// TwinCAT 3 PLC project PLC_Project
// ProgramVersion: 3.1.4024.0
// libraries:
//   Tc2_ControllerToolbox, * (Beckhoff Automation GmbH)
//   Tc2_Standard, * (Beckhoff Automation GmbH)
//   Tc2_System, * (Beckhoff Automation GmbH)
//   Tc2_TempController, * (Beckhoff Automation GmbH)
//   Tc3_Module, * (Beckhoff Automation GmbH)
//   VisuSymbols,3.5.10.0,System
// project tree:
//   / GlobalTextList.TcGTLO, PlcTask.TcTTO
//   GVLs/ Plant_Variables.TcGVL
//   POUs/Function Blocks/Control Valve Function Block/ Control_Valve.TcPOU, PID_Modes.TcDUT
//   POUs/Function Blocks/Pressure Transducer Function Block/ Pressure_Transducer.TcPOU
//   POUs/ MAIN.TcPOU
//   VISUs/ Tank_Visualization.TcVIS, VisualizationManager.TcVMO (not stored)
// real-time tasks:
//   TASK PlcTask: cycle T#10ms, priority 20, ADS port 350

CONFIGURATION PLC_Project
    RESOURCE PLC ON TwinCAT3
        TASK PlcTask(INTERVAL := T#10ms, PRIORITY := 20);
        PROGRAM MAIN WITH PlcTask : MAIN;
    END_RESOURCE
END_CONFIGURATION

// ---- POUs/Function Blocks/Control Valve Function Block/PID_Modes.TcDUT
{attribute 'qualified_only'}
{attribute 'strict'}
TYPE PID_Modes :
(
	Manual 		:= 	0,
	Automatic	:=	1
);
END_TYPE

// ---- GVLs/Plant_Variables.TcGVL
//{attribute 'qualified_only'}
VAR_GLOBAL
	Tank_Pressure			:	Pressure_Transducer;
	Input_Control_Valve		:	Control_Valve;
END_VAR

// ---- POUs/MAIN.TcPOU
PROGRAM MAIN
VAR
	Required_Tank_Pressure				:	REAL	:=	250.00;		//	kPa(a)	
	Simulated_Pressure_From_IO_Card		:	INT		:=	0;			//	4mA
	
	fInflowRate							:	LREAL	:=	0.0;
	fOutflowRate						:	LREAL	:=	2500;		//	Assume A Constant Drain To Feed Plant Equipment
	
	RandomFlowGenerator					:	FB_CTRL_NOISE_GENERATOR;	
	NoiseGeneratorMode					: 	E_CTRL_MODE						:=	E_CTRL_MODE.eCTRL_MODE_ACTIVE;
	NoiseSignal							: 	LREAL;
	RandomFlowGeneratorState			: 	Tc2_ControllerToolbox.E_CTRL_STATE;
	RandomFlowGeneratorErrorId			: 	Tc2_ControllerToolbox.E_CTRL_ERRORCODES;
	RandomFlowGeneratorErrorDetected	: 	BOOL;
	RandomFlowGeneratorParameters		: 	ST_CTRL_NOISE_GENERATOR_PARAMS;
END_VAR

{Region	"Read Tanks Pressure Transducer"}
Tank_Pressure(Input_mA	:=	Simulated_Pressure_From_IO_Card);
{endregion}

{Region "Perform PID Control On Input Control Valve"}
Input_Control_Valve(Controller_Setpoint					:=	Required_Tank_Pressure,
					Current_Process_Variable_Setpoint	:=	Tank_Pressure.Input_SI,
					Manual_Automatic_Mode				:=	PID_Modes.Automatic);
{endregion}

{Region "Random Flow Generator"}
//	Generate Some Gaussian Noise To Simulate PID Control Through Disturbances
RandomFlowGeneratorParameters.fAmplitude		:=	1000.0;
RandomFlowGeneratorParameters.tCtrlCycleTime	:=	T#10MS;
RandomFlowGeneratorParameters.tTaskCycleTime	:=	T#10MS;

RandomFlowGenerator(fManSyncValue	:=	20.0,
					eMode			:=	NoiseGeneratorMode,
					fOut			=>	NoiseSignal,
					eState			=>	RandomFlowGeneratorState,
					eErrorId		=>	RandomFlowGeneratorErrorId,
					bError			=>	RandomFlowGeneratorErrorDetected,
					stParams		:=	RandomFlowGeneratorParameters);
	
{endregion}

{Region "Simulate Field Input"}
// Simulate inflow proportional to valve position
fInflowRate := Input_Control_Valve.HMI_Valve_Reference * 330.0; // Max 10 kPa/sec new 300

// Update tank pressure
Simulated_Pressure_From_IO_Card := LREAL_TO_INT(Simulated_Pressure_From_IO_Card*0.05 + (fInflowRate - fOutflowRate)(* * 0.01*)) + LREAL_TO_INT(NoiseSignal); // 10 ms Cycle Implemented
{endregion}

END_PROGRAM

// ---- POUs/Function Blocks/Pressure Transducer Function Block/Pressure_Transducer.TcPOU
FUNCTION_BLOCK Pressure_Transducer
VAR_INPUT
	Input_mA						:	INT		:=	0;		//	Field Input Whereby 4 - 20mA Will Be Read As A 0 - 32768 Value From I/O Card
	Sensor_Minimum_SI_Measurement	:	REAL	:=	0.000;	//	kPa (a)
	Sensor_Maximum_SI_Measurement	:	REAL	:=	500.0;	//	kPa (a)
	
	//	Alarm Setpoints
	High_Alarm_Setpoint				:	REAL	:=	480.0;	//	kPa(a)
	Low_Alarm_Setpoint				:	REAL	:= 	87.00;	//	Kpa(a) @ Atmosphere
END_VAR
VAR_OUTPUT
	Input_SI						:	lREAL	:=	0.0;	//	Field Input In SI units
	
	//	Alarming 
	ScalingErrorDetected			: 	BOOL	:=	FALSE;
	High_Alarm						:	BOOL	:=	FALSE;
	Low_Alarm						:	BOOL	:=	FALSE;
END_VAR
VAR
	Field_Measurement_Scaler		:	FB_CTRL_SCALE;		//	Function To Scale 4 - 20mA To 0 - 500kPa Measurement
	ScalingErrorId					:	E_CTRL_ERRORCODES;
	ScalingParameters				: 	ST_CTRL_SCALE_PARAMS;
END_VAR

{Region "Scaling Setpoints"}
ScalingParameters.fInMin				:=		0;
ScalingParameters.fInMax				:=		32768;	//	16-Bit Analogue Input Card Maximum Reading (EL3024)
ScalingParameters.fOutMin				:=		Sensor_Minimum_SI_Measurement;	//	kPa
ScalingParameters.fOutMax				:=		Sensor_Maximum_SI_Measurement;	//	kPa
ScalingParameters.tCtrlCycleTime		:=		T#10MS;
ScalingParameters.tTaskCycleTime		:=		T#10MS;
{endregion}

{Region "Scale Input To SI Value"}
Field_Measurement_Scaler(	fIn			:=	Input_mA,
							fOut		=>	Input_SI,
							eErrorId	=>	ScalingErrorId,
							bError		=>	ScalingErrorDetected,
							stParams	:=	ScalingParameters);
{endregion}							
							
{region "Alarm_Detection"}
//	Low Alarm Functionality: Single Shot Pulse Will Set An Event In The Event Manager
IF(Input_SI <= Low_Alarm_Setpoint)THEN
	Low_Alarm	:=	TRUE;
ELSE
	Low_Alarm	:=	FALSE;		 
END_IF;
	 
//	High Alarm Functionality Single Shot Pulse Will Set An Event In The Event Manager
IF(Input_SI >= High_Alarm_Setpoint)THEN
	High_Alarm	:=	TRUE;
ELSE
	High_Alarm	:=	FALSE;		 
END_IF;		  
{endregion}						

{Region "Trend Generation"}

{endregion}

END_FUNCTION_BLOCK

// ---- POUs/Function Blocks/Control Valve Function Block/Control_Valve.TcPOU
FUNCTION_BLOCK Control_Valve
VAR_INPUT
	Controller_Setpoint					: 	LREAL 		:= 	0.0;
	Current_Process_Variable_Setpoint	:	LREAL 		:=	0.0;
	Operator_Set_PID_Output_Value		: 	LREAL 		:= 	0.0;
	
	// PID Gains & Setpoints
	Proportional_Gain					:	REAL		:=	3.0;
	Integral_Gain						:	TIME		:=	T#1S;
	Derivative_Gain						:	TIME		:=	T#0.25S;
	Damping_Time						:	TIME		:=	T#0.1S;
	Minimum_Output_Value				:	REAL		:=	0.0;
	Maximum_Output_Value				:	REAL		:=	32768.0;
	
	//	PID Mode Selection
	Manual_Automatic_Mode				:	INT			:=	PID_Modes.Automatic;
END_VAR
VAR_OUTPUT
	IO_Valve_Reference					:	INT			:=	0;
	HMI_Valve_Reference					:	LREAL		:=	0.0;
	Error_Detected						: 	BOOL 		:= 	FALSE;
END_VAR
VAR
	PID_Controller						:	FB_CTRL_PID;
	
	// Used For Bumpless Transfer Between Automatic & Manual Modes Of PID Controller.
	bSync								: 	BOOL		:= FALSE;
	PID_Controller_Mode: E_CTRL_MODE 	:= 	E_CTRL_MODE.eCTRL_MODE_IDLE;
	Controller_Valve_Reference			:	LREAL		:=	0;
	Hold_Output							: 	BOOL;
	Restrict_Controller_Output			: 	BOOL;
	Current_Controller_State			:	E_CTRL_STATE;
	Error_Code							:	E_CTRL_ERRORCODES;
	PID_Control_Parameters				:	ST_CTRL_PID_PARAMS;
	
	//	Output Scaling To HMI Visualisation
	Output_Scaler						:	FB_CTRL_SCALE;
	ScalingParameters					: 	ST_CTRL_SCALE_PARAMS;
	ScalingErrorId						:	E_CTRL_ERRORCODES;
	ScalingErrorDetected				: 	BOOL	:=	FALSE;
END_VAR

{Region "PID Initialization"}
PID_Control_Parameters.tCtrlCycleTime	:=	T#10MS;	
PID_Control_Parameters.tTaskCycleTime	:=	T#10MS;	
PID_Control_Parameters.fKp				:=	Proportional_Gain;
PID_Control_Parameters.tTn				:=	Integral_Gain;
PID_Control_Parameters.tTv				:=	Derivative_Gain;
PID_Control_Parameters.tTd				:=	Damping_Time;
PID_Control_Parameters.fOutMinLimit		:=	Minimum_Output_Value;
PID_Control_Parameters.fOutMaxLimit		:=	Maximum_Output_Value;
{endregion}

{Region "PID Mode Selection"}
IF(Manual_Automatic_Mode    = PID_Modes.Manual)THEN
	PID_Controller_Mode					:=	E_CTRL_MODE.eCTRL_MODE_MANUAL;
ELSIF(Manual_Automatic_Mode = PID_Modes.Automatic)THEN
	PID_Controller_Mode					:=	E_CTRL_MODE.eCTRL_MODE_ACTIVE;
ELSE
	PID_Controller_Mode					:=	E_CTRL_MODE.eCTRL_MODE_IDLE;
END_IF
{endregion}

{Region "PID Control"}
PID_Controller(	fSetpointValue			:=	Controller_Setpoint,
				fActualValue			:=	Current_Process_Variable_Setpoint,
				fManSyncValue			:=	Operator_Set_PID_Output_Value,
				bSync					:=	bSync,
				eMode					:=	PID_Controller_Mode,
				bHold					:=	Hold_Output,
				fOut					=>	Controller_Valve_Reference,
				bARWactive				=>	Restrict_Controller_Output,
				eState					=>	Current_Controller_State,
				eErrorId				=>	Error_Code,
				bError					=>	Error_Detected,
				stParams				:=	PID_Control_Parameters);
				
IO_Valve_Reference						:=	LREAL_TO_INT(Controller_Valve_Reference);	
{endregion}

{Region "PID Output Scaling"}
ScalingParameters.fInMin				:=		0;
ScalingParameters.fInMax				:=		32768;	//	16-Bit Analogue Input Card Maximum Reading (EL3024)
ScalingParameters.fOutMin				:=		0;		//	%
ScalingParameters.fOutMax				:=		100.0;	//	%
ScalingParameters.tCtrlCycleTime		:=		T#10MS;
ScalingParameters.tTaskCycleTime		:=		T#10MS;

Output_Scaler(				fIn			:=	Controller_Valve_Reference,
							fOut		=>	HMI_Valve_Reference,
							eErrorId	=>	ScalingErrorId,
							bError		=>	ScalingErrorDetected,
							stParams	:=	ScalingParameters);
{endregion}

END_FUNCTION_BLOCK

// ---- GlobalTextList.TcGTLO
TEXTLIST GlobalTextList
  496 = '%'
  337 = '%5.2f'
  527 = '%s'
  362 = 'Actual Pressure'
  93 = 'Buffer Tank'
  791 = 'Control Valve'
  587 = 'Input'
  111 = 'kPa(a)'
  178 = 'Output'
  782 = 'Setpoint'
END_TEXTLIST

// ---- VISUs/Tank_Visualization.TcVIS
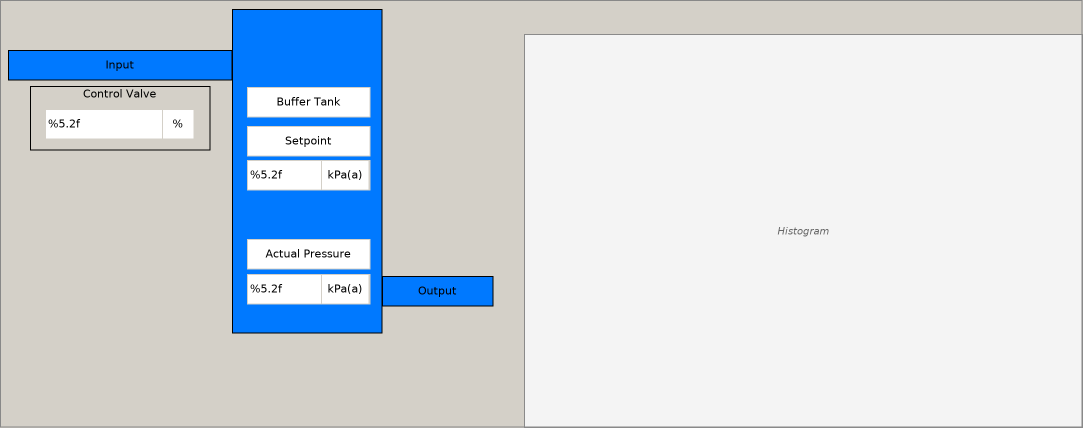
VISUALIZATION Tank_Visualization  // 1083x428
    RoundedRectangle (30,86 180x64), "Control Valve"
    RoundedRectangle (232,9 150x324)
    Rectangle (382,276 111x30), "Output"
    Rectangle (8,50 224x30), "Input"
    Textfield (247,87 123x30), "Buffer Tank"
    Textfield (45,109 150x30), "%5.2f", text variable: Input_Control_Valve.HMI_Valve_Reference
    Textfield (247,274 123x30), "%5.2f", text variable: Tank_Pressure.Input_SI
    Textfield (321,274 48x30), "kPa(a)"
    Textfield (162,109 32x30), "%"
    Textfield (247,160 123x30), "%5.2f", text variable: Input_Control_Valve.Controller_Setpoint
    Textfield (321,160 48x30), "kPa(a)"
    Textfield (247,126 123x30), "Setpoint"
    Textfield (247,239 123x30), "Actual Pressure"
    Histogram (524,34 559x394), scale format: %.1f, scale 0..500
END_VISUALIZATION
